FUNCTION_BLOCK FB_Module
VAR_INPUT
END_VAR
VAR_OUTPUT
END_VAR
VAR
END_VAR

END_FUNCTION_BLOCK

(* stored: Version 1.1.0.1, ProductVersion 3.1.4024.4
   POU FB_Module: Id {b6184298-8309-4406-9099-e98708c7ef5d}, SpecialFunc None *)
